Fanuc KAREL source: ka00130.KL

-- PROVISIONAL review KL for V940-1; original PC SHA256 54d6b5a0488ed36e515abeb794a803a9fba23f6d72452ffb947e8d0af9149d8d
-- Incomplete behavior may be omitted. Consult companion uncertainty JSON. Do not deploy.
PROGRAM KA00130
%NOLOCKGROUP
-- UNRESOLVED_DECL SRC type=002018
-- UNRESOLVED_DECL DST type=00001c
BEGIN
  -- V9_ZERO_TABLE_METADATA_HINT layout=0001; no indexed target words; source/name/runtime held
  -- UNRESOLVED_PC offsets 5-19; opcodes 2E,22,9D,33,B2
  -- UNRESOLVED_PC offsets 24-39; opcodes 22,9D,33,B1,23
  -- UNRESOLVED_PC offsets 44-48; opcodes 7F
END KA00130
